(* Logix 5000 project; controller R1USB70001_CWRU_Scenario_Gen_20111116 vendor 1 type 14 code 54 rev 19.11; software revision 19.01; part 9 of 9 *)
(* tags used below, declared in another part *)
   EditScenario : EditScenarioPub;
   Execute : ExecutePub;
   HMI : HMIPub;
(* MainProgram, continued *)

ROUTINE MainRoutine   (* ladder *)
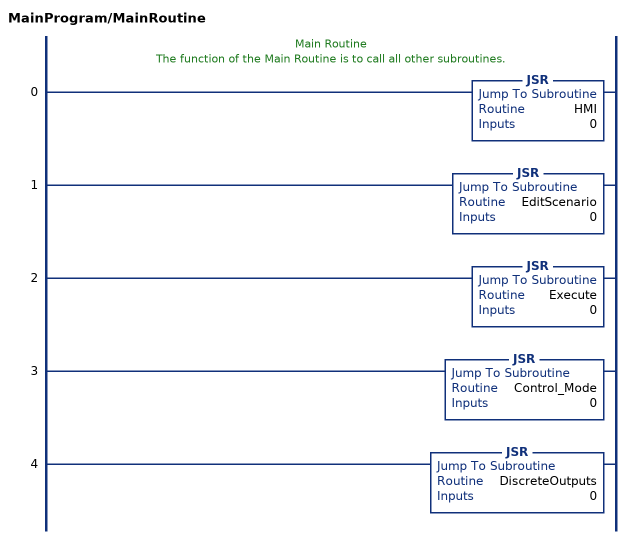
   // Main Routine
   // The function of the Main Routine is to call all other subroutines.
   0: JSR(HMI,0);
   1: JSR(EditScenario,0);
   2: JSR(Execute,0);
   3: JSR(Control_Mode,0);
   4: JSR(DiscreteOutputs,0);
END_ROUTINE
END_PROGRAM
